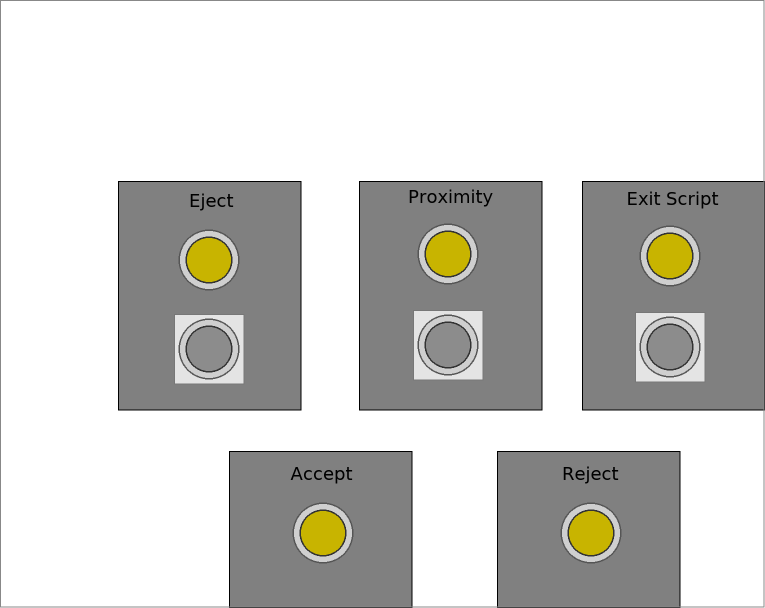
VISUALIZATION HMI  // 765x608
    RoundedRectangle (359,181 183x229)
    PushSwitch (413,310 70x70), variable: LadderLogicBottleChecker.ProximitySensor, behaviour: TOGGLE, style: Switch-PushSwitch-Gray
    Lamp1 (413,219 70x70), variable: LadderLogicBottleChecker.ProximitySensor, style: Lamp-Lamp1-Yellow
    Rectangle (376,183 149x28), "Proximity"
    RoundedRectangle (582,181 183x229)
    PushSwitch (635,312 70x70), variable: LadderLogicBottleChecker.ExitScript, behaviour: TOGGLE, style: Switch-PushSwitch-Gray
    Lamp1 (635,221 70x70), variable: LadderLogicBottleChecker.ExitScript, style: Lamp-Lamp1-Yellow
    Rectangle (598,185 149x28), "Exit Script"
    RoundedRectangle (118,181 183x229)
    PushSwitch (174,314 70x70), variable: LadderLogicBottleChecker.EjectBottle, behaviour: TOGGLE, style: Switch-PushSwitch-Gray
    Lamp1 (174,225 70x70), variable: LadderLogicBottleChecker.EjectRelay, style: Lamp-Lamp1-Yellow
    Rectangle (137,187 149x28), "Eject"
    RoundedRectangle (229,451 183x157)
    Rectangle (247,460 149x28), "Accept"
    RoundedRectangle (497,451 183x157)
    Rectangle (516,460 149x28), "Reject"
    Lamp1 (556,498 70x70), variable: LadderLogicBottleChecker.RejectFlag, style: Lamp-Lamp1-Yellow
    Lamp1 (288,498 70x70), variable: LadderLogicBottleChecker.AcceptFlag, style: Lamp-Lamp1-Yellow
END_VISUALIZATION

(* stored: Version 1.1.0.1, ProductVersion 3.1.4026.8
   Visu HMI: Id {2dae3e48-dc84-4f83-9aee-5bd7d7869ae8} *)
